(* IEC 61131-3 sources: Lasal/CPU_5344_V01/Class/dbSettings, 1 file *)

(* ---- dbSettings.st ---- *)
(*!
<Class
	Name               = "dbSettings"
	Revision           = "0.0"
	RealtimeTask       = "false"
	CyclicTask         = "false"
	BackgroundTask     = "false"
	Sigmatek           = "false"
	OSInterface        = "false"
	HighPriority       = "false"
	Automatic          = "false"
	UpdateMode         = "Prescan"
	SharedCommandTable = "true"
	Objectsize         = "(750,1140)">
	<Channels>
		<Server Name="allWasteAtFront" Visualized="true" Initialize="false" WriteProtected="false" Retentive="File"/>
		<Server Name="AutoActive" Visualized="true" Initialize="false" WriteProtected="false" Retentive="File"/>
		<Server Name="ClassSvr" Visualized="false" Initialize="false" WriteProtected="true" Retentive="false"/>
		<Server Name="clsBU1" Visualized="true" Initialize="true" DefValue="0" WriteProtected="false" Retentive="File"/>
		<Server Name="clsBU10" Visualized="true" Initialize="false" WriteProtected="false" Retentive="File"/>
		<Server Name="clsBU2" Visualized="true" Initialize="true" WriteProtected="false" Retentive="File"/>
		<Server Name="clsBU3" Visualized="true" Initialize="true" WriteProtected="false" Retentive="File"/>
		<Server Name="clsBU4" Visualized="true" Initialize="false" WriteProtected="false" Retentive="File"/>
		<Server Name="clsBU5" Visualized="true" Initialize="false" WriteProtected="false" Retentive="File"/>
		<Server Name="clsBU6" Visualized="true" Initialize="false" WriteProtected="false" Retentive="File"/>
		<Server Name="clsBU7" Visualized="true" Initialize="false" WriteProtected="false" Retentive="File"/>
		<Server Name="clsBU8" Visualized="true" Initialize="false" WriteProtected="false" Retentive="File"/>
		<Server Name="clsBU9" Visualized="true" Initialize="false" WriteProtected="false" Retentive="File"/>
		<Server Name="combineOperations" Visualized="true" Initialize="false" WriteProtected="false" Retentive="File"/>
		<Server Name="doEndWaste" Visualized="true" Initialize="false" WriteProtected="false" Retentive="File"/>
		<Server Name="doFrontWaste" Visualized="true" Initialize="false" WriteProtected="false" Retentive="File"/>
		<Server Name="freeSpaceLoadMaterial" Visualized="true" Initialize="false" WriteProtected="false" Retentive="File"/>
		<Server Name="lengthBetweenPiece" Visualized="true" Initialize="false" WriteProtected="false" Retentive="File"/>
		<Server Name="lengthGripProfile" Visualized="true" Initialize="false" WriteProtected="false" Retentive="File"/>
		<Server Name="magazinPositionBigWaste" Visualized="true" Initialize="false" WriteProtected="false" Retentive="File"/>
		<Server Name="maxLengthForWasteBin" Visualized="true" Initialize="false" WriteProtected="false" Retentive="File"/>
		<Server Name="maxLengthWaste" Visualized="true" Initialize="false" WriteProtected="false" Retentive="File"/>
		<Server Name="maxPosCl1" Visualized="true" Initialize="false" WriteProtected="false" Retentive="File"/>
		<Server Name="maxPosCl2" Visualized="true" Initialize="false" WriteProtected="false" Retentive="File"/>
		<Server Name="maxPosCl3" Visualized="true" Initialize="false" WriteProtected="false" Retentive="File"/>
		<Server Name="maxPosCl4" Visualized="true" Initialize="false" WriteProtected="false" Retentive="File"/>
		<Server Name="maxPosCl5" Visualized="true" Initialize="false" WriteProtected="false" Retentive="File"/>
		<Server Name="maxPosCl6" Visualized="true" Initialize="false" WriteProtected="false" Retentive="File"/>
		<Server Name="maxPosCl7" Visualized="true" Initialize="false" WriteProtected="false" Retentive="File"/>
		<Server Name="maxPosCl8" Visualized="true" Initialize="false" WriteProtected="false" Retentive="File"/>
		<Server Name="maxPosCl9" Visualized="true" Initialize="false" WriteProtected="false" Retentive="File"/>
		<Server Name="maxTakeOverPos" Visualized="true" Initialize="false" WriteProtected="false" Retentive="File"/>
		<Server Name="minEndWaste" Visualized="true" Initialize="false" WriteProtected="false" Retentive="File"/>
		<Server Name="minEndWasteAngle" Visualized="true" Initialize="false" WriteProtected="false" Retentive="File"/>
		<Server Name="minFrontWaste" Visualized="true" Initialize="false" WriteProtected="false" Retentive="File"/>
		<Server Name="minLengthForOutputMagazines" Visualized="true" Initialize="false" WriteProtected="false" Retentive="File"/>
		<Server Name="minLengthProdInGripperX2" Visualized="true" Initialize="false" WriteProtected="false" Retentive="File"/>
		<Server Name="minLengthRollersOutputWithoutMove" Visualized="true" Initialize="false" WriteProtected="false" Retentive="File"/>
		<Server Name="minPosCl1" Visualized="true" Initialize="false" WriteProtected="false" Retentive="File"/>
		<Server Name="minPosCl2" Visualized="true" Initialize="false" WriteProtected="false" Retentive="File"/>
		<Server Name="minPosCl3" Visualized="true" Initialize="false" WriteProtected="false" Retentive="File"/>
		<Server Name="minPosCl4" Visualized="true" Initialize="false" WriteProtected="false" Retentive="File"/>
		<Server Name="minPosCl5" Visualized="true" Initialize="false" WriteProtected="false" Retentive="File"/>
		<Server Name="minPosCl6" Visualized="true" Initialize="false" WriteProtected="false" Retentive="File"/>
		<Server Name="minPosCl7" Visualized="true" Initialize="false" WriteProtected="false" Retentive="File"/>
		<Server Name="minPosCl8" Visualized="true" Initialize="false" WriteProtected="false" Retentive="File"/>
		<Server Name="minPosCl9" Visualized="true" Initialize="false" WriteProtected="false" Retentive="File"/>
		<Server Name="minPosLeftSawClampClosed" Visualized="true" Initialize="false" WriteProtected="false" Retentive="File"/>
		<Server Name="minPosWagonUp" Visualized="true" Initialize="false" WriteProtected="false" Retentive="File"/>
		<Server Name="minTakeOverPos" Visualized="true" Initialize="false" WriteProtected="false" Retentive="File"/>
		<Server Name="moveBigWasteToMagazin" Visualized="true" Initialize="false" WriteProtected="false" Retentive="File"/>
		<Server Name="noWasteStop" Visualized="true" Initialize="false" WriteProtected="false" Retentive="File"/>
		<Server Name="offsetBu3" Visualized="true" Initialize="false" WriteProtected="false" Retentive="File"/>
		<Server Name="offsetBu6" Visualized="true" Initialize="false" WriteProtected="false" Retentive="File"/>
		<Server Name="offsetBu7" Visualized="true" Initialize="false" WriteProtected="false" Retentive="File"/>
		<Server Name="offsetOutput" Visualized="true" Initialize="false" WriteProtected="false" Retentive="File"/>
		<Server Name="offsetPressureRol" Visualized="true" Initialize="false" WriteProtected="false" Retentive="File"/>
		<Server Name="offsetTakeIn" Visualized="true" Initialize="false" WriteProtected="false" Retentive="File"/>
		<Server Name="offsetWasteStop" Visualized="true" Initialize="false" WriteProtected="false" Retentive="File"/>
		<Server Name="openPressureRollAtFirstOperation" Visualized="true" Initialize="false" WriteProtected="false" Retentive="File"/>
		<Server Name="optimumTakeOverPos" Visualized="true" Initialize="false" WriteProtected="false" Retentive="File"/>
		<Server Name="overTakeActive" Visualized="true" Initialize="true" DefValue="0" WriteProtected="false" Retentive="File"/>
		<Server Name="parMaxForceWagonX1" Visualized="true" Initialize="false" WriteProtected="false" Retentive="File"/>
		<Server Name="pushMaterialToMinPos" Visualized="true" Initialize="false" WriteProtected="false" Retentive="File"/>
		<Server Name="safeDistanceToMaterialMill" Visualized="true" Initialize="false" WriteProtected="false" Retentive="File"/>
		<Server Name="sawWidth" Visualized="true" Initialize="false" WriteProtected="false" Retentive="File"/>
		<Server Name="slowXSpeed" Visualized="true" Initialize="false" WriteProtected="false" Retentive="File"/>
		<Server Name="speedDrill1" Visualized="true" Initialize="false" WriteProtected="false" Retentive="File"/>
		<Server Name="speedDrill2" Visualized="true" Initialize="false" WriteProtected="false" Retentive="File"/>
		<Server Name="speedDrill3" Visualized="true" Initialize="false" WriteProtected="false" Retentive="File"/>
		<Server Name="speedDrill4" Visualized="true" Initialize="false" WriteProtected="false" Retentive="File"/>
		<Server Name="toolDiamMill1" Visualized="true" Initialize="false" WriteProtected="false" Retentive="File"/>
		<Server Name="toolDiamMill2" Visualized="true" Initialize="false" WriteProtected="false" Retentive="File"/>
		<Server Name="toolDiamMill3" Visualized="true" Initialize="false" WriteProtected="false" Retentive="File"/>
		<Server Name="toolDiamMill4" Visualized="true" Initialize="false" WriteProtected="false" Retentive="File"/>
		<Server Name="toolLengthMill1" Visualized="true" Initialize="false" WriteProtected="false" Retentive="File"/>
		<Server Name="toolLengthMill2" Visualized="true" Initialize="false" WriteProtected="false" Retentive="File"/>
		<Server Name="toolLengthMill3" Visualized="true" Initialize="false" WriteProtected="false" Retentive="File"/>
		<Server Name="toolLengthMill4" Visualized="true" Initialize="false" WriteProtected="false" Retentive="File"/>
		<Server Name="usedUnitsCl1" Visualized="true" Initialize="true" DefValue="6" WriteProtected="false" Retentive="File"/>
		<Server Name="usedUnitsCl2" Visualized="true" Initialize="false" WriteProtected="false" Retentive="File"/>
		<Server Name="usedUnitsCl3" Visualized="true" Initialize="false" WriteProtected="false" Retentive="File"/>
		<Server Name="usedUnitsCl4" Visualized="true" Initialize="false" WriteProtected="false" Retentive="File"/>
		<Server Name="usedUnitsCl5" Visualized="true" Initialize="false" WriteProtected="false" Retentive="File"/>
		<Server Name="usedUnitsCl6" Visualized="true" Initialize="false" WriteProtected="false" Retentive="File"/>
		<Server Name="usedUnitsCl7" Visualized="true" Initialize="false" WriteProtected="false" Retentive="File"/>
		<Server Name="usedUnitsCl8" Visualized="true" Initialize="false" WriteProtected="false" Retentive="File"/>
		<Server Name="usedUnitsCl9" Visualized="true" Initialize="false" WriteProtected="false" Retentive="File"/>
		<Server Name="usePressureRoll" Visualized="true" Initialize="false" WriteProtected="false" Retentive="File"/>
		<Server Name="waitPosX2" Visualized="true" Initialize="false" WriteProtected="false" Retentive="File"/>
		<Server Name="wasteStopForEndWaste" Visualized="true" Initialize="true" DefValue="0" WriteProtected="false" Retentive="File"/>
		<Server Name="widthBu6" Visualized="false" Initialize="true" DefValue="650" WriteProtected="false" Retentive="false"/>
		<Server Name="workingXSpeed" Visualized="true" Initialize="false" WriteProtected="false" Retentive="File"/>
	</Channels>
</Class>
*)
dbSettings : CLASS
  //Servers:
	ClassSvr 	: SvrChCmd_DINT;
	sawWidth 	: SvrCh_DINT;
	wasteStopForEndWaste 	: SvrCh_DINT;
	maxLengthWaste 	: SvrCh_DINT;
	allWasteAtFront 	: SvrCh_DINT;
	overTakeActive 	: SvrCh_DINT;
	minFrontWaste 	: SvrCh_DINT;
	minEndWaste 	: SvrCh_DINT;
	minEndWasteAngle 	: SvrCh_DINT;
	doFrontWaste 	: SvrCh_DINT;
	doEndWaste 	: SvrCh_DINT;
	noWasteStop 	: SvrCh_DINT;
	lengthBetweenPiece 	: SvrCh_DINT;
	moveBigWasteToMagazin 	: SvrCh_DINT;
	magazinPositionBigWaste 	: SvrCh_DINT;
	freeSpaceLoadMaterial 	: SvrCh_DINT;
	lengthGripProfile 	: SvrCh_DINT;
	minLengthProdInGripperX2 	: SvrCh_DINT;
	optimumTakeOverPos 	: SvrCh_DINT;
	combineOperations 	: SvrCh_DINT;
	minTakeOverPos 	: SvrCh_DINT;
	maxTakeOverPos 	: SvrCh_DINT;
	offsetTakeIn 	: SvrCh_DINT;
	offsetWasteStop 	: SvrCh_DINT;
	offsetOutput 	: SvrCh_DINT;
	waitPosX2 	: SvrCh_DINT;
	minLengthForOutputMagazines 	: SvrCh_DINT;
	workingXSpeed 	: SvrCh_DINT;
	slowXSpeed 	: SvrCh_DINT;
	minPosWagonUp 	: SvrCh_DINT;
	minPosLeftSawClampClosed 	: SvrCh_DINT;
	minLengthRollersOutputWithoutMove 	: SvrCh_DINT;
	offsetBu3 	: SvrCh_DINT;
	offsetBu6 	: SvrCh_DINT;
	widthBu6 	: SvrCh_DINT;
	offsetBu7 	: SvrCh_DINT;
	minPosCl1 	: SvrCh_DINT;
	maxPosCl1 	: SvrCh_DINT;
	usedUnitsCl1 	: SvrCh_Units;
	minPosCl2 	: SvrCh_DINT;
	maxPosCl2 	: SvrCh_DINT;
	usedUnitsCl2 	: SvrCh_Units;
	minPosCl3 	: SvrCh_DINT;
	maxPosCl3 	: SvrCh_DINT;
	usedUnitsCl3 	: SvrCh_Units;
	minPosCl4 	: SvrCh_DINT;
	maxPosCl4 	: SvrCh_DINT;
	usedUnitsCl4 	: SvrCh_Units;
	minPosCl5 	: SvrCh_DINT;
	maxPosCl5 	: SvrCh_DINT;
	usedUnitsCl5 	: SvrCh_Units;
	minPosCl6 	: SvrCh_DINT;
	maxPosCl6 	: SvrCh_DINT;
	usedUnitsCl6 	: SvrCh_Units;
	minPosCl7 	: SvrCh_DINT;
	maxPosCl7 	: SvrCh_DINT;
	usedUnitsCl7 	: SvrCh_Units;
	minPosCl8 	: SvrCh_DINT;
	maxPosCl8 	: SvrCh_DINT;
	usedUnitsCl8 	: SvrCh_Units;
	minPosCl9 	: SvrCh_DINT;
	maxPosCl9 	: SvrCh_DINT;
	usedUnitsCl9 	: SvrCh_Units;
	clsBU1 	: SvrCh_Units;
	clsBU2 	: SvrCh_Units;
	clsBU3 	: SvrCh_Units;
	clsBU4 	: SvrCh_Units;
	clsBU5 	: SvrCh_Units;
	clsBU6 	: SvrCh_Units;
	clsBU7 	: SvrCh_Units;
	clsBU8 	: SvrCh_Units;
	clsBU9 	: SvrCh_Units;
	clsBU10 	: SvrCh_Units;
	toolDiamMill1 	: SvrCh_DINT;
	toolDiamMill2 	: SvrCh_DINT;
	toolDiamMill3 	: SvrCh_DINT;
	toolDiamMill4 	: SvrCh_DINT;
	speedDrill1 	: SvrCh_DINT;
	speedDrill2 	: SvrCh_DINT;
	speedDrill3 	: SvrCh_DINT;
	speedDrill4 	: SvrCh_DINT;
	toolLengthMill1 	: SvrCh_DINT;
	toolLengthMill2 	: SvrCh_DINT;
	toolLengthMill3 	: SvrCh_DINT;
	toolLengthMill4 	: SvrCh_DINT;
	safeDistanceToMaterialMill 	: SvrCh_DINT;
	usePressureRoll 	: SvrCh_DINT;
	openPressureRollAtFirstOperation 	: SvrCh_DINT;
	pushMaterialToMinPos 	: SvrCh_DINT;
	offsetPressureRol 	: SvrCh_DINT;
	maxLengthForWasteBin 	: SvrCh_DINT;
	AutoActive 	: SvrCh_DINT;
	parMaxForceWagonX1 	: SvrCh_DINT;
  //Clients:
  //Variables:
  //Functions:
  //Tables:
	FUNCTION @STD
		VAR_OUTPUT
			ret_code	: CONFSTATES;
		END_VAR;
	FUNCTION GLOBAL TAB @CT_;
END_CLASS;
